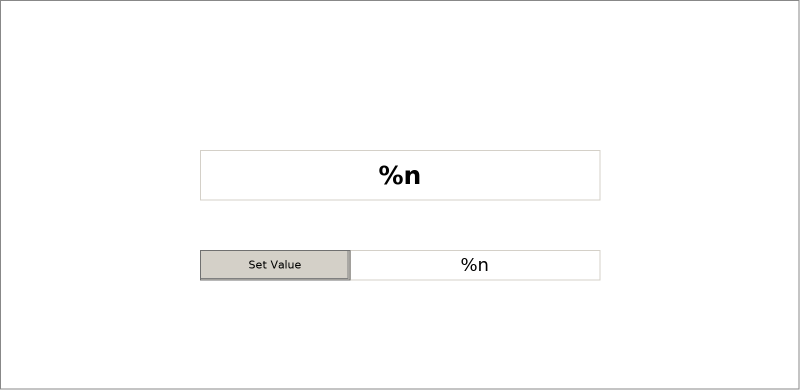
VISUALIZATION VisuKL5151Control  // 800x390
VAR_IN_OUT
	pDev : POINTER TO FB_DevKL5151;
END_VAR
    Textfield (200,150 400x50), "%n", text variable: pDev^.stManualControl.nCount
    Textfield (350,250 250x30), "%n", text variable: pDev^.stManualControl.nManValue
        OnMouseClick: write the text variable via VisuDialogs.Numpad
    Button (200,250 150x30), "Set Value"
        tap pDev^.stManualControl.bManSetValue
END_VISUALIZATION

(* stored: Version 1.1.0.1, ProductVersion 3.1.4024.11
   Visu VisuKL5151Control: Id {34b3a67e-d41c-0434-0164-f2ca240b679f} *)
